Universal Robots PolyScope program: followeroptTFM.urp

Program followeroptTFM (installation=default directory=/home/ur/ursim-current/programs createdIn=3.5.4.10845 lastSavedIn=3.13.0.10253 robotSerialNumber=2018339999)
Calibrated DH parameters: a=[0, -0.24355, -0.2132, 0, 0, 0]; d=[0.15185, 0, 0, 0.13105, 0.08535, 0.0921]; alpha=[1.570796, 0, 0, 1.570796, -1.570796, 0]; deltaTheta=[0, 0, 0, 0, 0, 0]
BeforeStart
  t := 0.008
  look_ahead := 0.2
  gain := 100
  samejoints := 0
  start := False
  initdif := d2r(1.5)
  diffang := [initdif,initdif,initdif,initdif,initdif,initdif]
  newjoints := [255.0,255.0,255.0,255.0,255.0,255.0]
  mb_o_regfol := [255.0,255.0,255.0,255.0,255.0,255.0]
  mb_o_regown := [255.0,255.0,255.0,255.0,255.0,255.0]
  mb_o_regfol_rev := [255.0,255.0,255.0,255.0,255.0,255.0]
  Script: sync()
  Call get_master_q
  'If the connection with the master it's right the vale is different from the initialized value'
  If newjoints≠[255.0,255.0,255.0,255.0,255.0,255.0]
    MoveJ speed 60 deg/s, acceleration 80 deg/s^2 (useActiveTCP=true)
      Waypoint Waypoint (Variable): variable=newjoints
  Else 
    Popup Message (haltProgram=false message=Can not connect with the master inputType=Text)
    Halt
Robot Program (runOnlyOnce=false)
  'Moves the robot'
  Script: servoj(newjoints,t=t,lookahead_time=look_ahead,gain=gain)
Thread Subproceso_1 (runOnlyOnce=false)
  Folder Master joints
    mb_o_regfol := [j0,j1,j2,j3,j4,j5]
    mb_o_regfol_rev := [r0,r1,r2,r2,r4,r5]
  Calc := 0
  Loop While (checkContinuously=false) expression=Calc<6
    Script: mb_o_regfol[Calc]=mb_o_regfol[Calc]/1000
    If mb_o_regfol_rev[Calc]≥1
      Script: mb_o_regfol[Calc]=-1*(6.283-mb_o_regfol[Calc])
    Script: diffang[Calc]=mb_o_regfol[Calc]-mb_o_regown[Calc]
    SuppressedNode
      newjoints := mb_o_regfol
    Calc := Calc+1
  newjoints := mb_o_regfol
  Script: sync()
Thread Thread_1 (runOnlyOnce=false)
  'Get my joint angles'
  mb_o_regown := get_actual_joint_positions()
  'Get the master angles'
  Call get_master_q
  Script: sync()
SubProgram -> get_master_q
SubProgram get_master_q (keepSynchronizedWithDisk=false)
  Folder Master joints
    'Joints of the master'
    mb_o_regfol := [j0,j1,j2,j3,j4,j5]
    'Revolutions of the master'
    mb_o_regfol_rev := [r0,r1,r2,r2,r4,r5]
  Calc := 0
  'Having the joint values and the revolutions of the master, I compute the follower ones'
  Loop While (checkContinuously=false) expression=Calc<6
    'Convert the data from mm to meters'
    Script: mb_o_regfol[Calc]=mb_o_regfol[Calc]/1000
    'Check the revolution sign'
    If mb_o_regfol_rev[Calc]≥1
      'If the revolution sign it's different from 0, modbus provides the complementary angle'
      Script: mb_o_regfol[Calc]=-1*(6.283-mb_o_regfol[Calc])
    'Computes the difference of angle between the master and the follower'
    Script: diffang[Calc]=norm(mb_o_regfol[Calc]-mb_o_regown[Calc])
    'Check if the difference it's greater than certain value, to avoid to be too sensible'
    If diffang[Calc] ≥ initdif
      Script: newjoints[Calc] = mb_o_regfol[Calc]
    Calc := Calc+1
  SuppressedNode
    newjoints := mb_o_regfol
